Universal Robots URScript: movel02.script

# movel:
# Set tcp: ignore active tcp
# Tool speed : 250mm/s
# Tool acceleration : 1200mm/s2
# waypoint1: feature view, xyz-RxRyRz (radian), Joint positions (degree)
# stop at this point
# use shared parameters

def movel02():
  global _hidden_verificationVariable=0
  set_safety_mode_transition_hardness(1)
  set_gravity([0.0, 0.0, 9.82])
  set_target_payload(1.000000, [0.000000, 0.000000, 0.000000], [0.001539, 0.001539, 0.001539, 0.000000, 0.000000, 0.000000])
  set_tcp(p[0.0,0.0,0.0,0.0,0.0,0.0])
  set_standard_analog_input_domain(0, 1)
  set_standard_analog_input_domain(1, 1)
  set_tool_analog_input_domain(0, 1)
  set_tool_analog_input_domain(1, 1)
  set_analog_outputdomain(0, 0)
  set_analog_outputdomain(1, 0)
  set_input_actions_to_default()
  set_tool_communication(False, 115200, 0, 1, 1.5, 3.5)
  set_tool_output_mode(0)
  set_tool_digital_output_mode(0, 1)
  set_tool_digital_output_mode(1, 1)
  set_tool_voltage(0)
  step_count_31a1baac_9259_41ae_be3a_8e460796e033 = 0.0
  thread Step_Counter_Thread_04bcb5a2_3784_42e7_a1fa_b66500996017():
    while (True):
      step_count_31a1baac_9259_41ae_be3a_8e460796e033 = step_count_31a1baac_9259_41ae_be3a_8e460796e033 + 1.0
      sync()
    end
  end
  run Step_Counter_Thread_04bcb5a2_3784_42e7_a1fa_b66500996017()
  global Waypoint_1_p=p[-.136861537556, -.267180821738, .146971261118, -.001221359682, 3.116276528482, .038891915637]
  global Waypoint_1_q=[-1.6006999999999998, -1.7271, -2.2029999999999994, -0.8079999999999998, 1.5951, -0.030999999999999694]
  while (True):
    $ 1 "Robot Program"
    $ 2 "MoveL"
    $ 3 "Waypoint_1" "breakAfter"
    movel(pose_trans(Waypoint_1_p, get_tcp_offset()), a=1.2, v=0.25)
  end
end
